*)
{attribute 'reflection'} 
FUNCTION_BLOCK FB_Mitsubishi_MRJ4TM EXTENDS FB_LinkDataReal 
VAR_INPUT
	pControl			: PVOID; //Pocess data from fieldbus, 29 BYTES FROM FIELDBUS
	pStatus				: PVOID; //Pocess data to fieldbus, 41 BYTES FROM FIELDBUS		
	stControl	 		: ST_Mitsubishi_MRJ4TM_Control;
	stConfig			: ST_Mitsubishi_MRJ4TM_Config;
	bSTO 				: BOOL := TRUE;
END_VAR

VAR_OUTPUT
	stStatus 			: ST_Mitsubishi_MRJ4TM_Status;	
END_VAR

VAR		
	{attribute 'instance-path'} 
    {attribute 'noinit'} 
    _sPath 				: STRING;
	_fbStateMachine 	: FB_DS402_FSM;
	_fbEncoder 			: FB_Encoder;	
END_VAR

SUPER^();
InitRun();

GetControlData();
Cycle();
SetStatusData();

METHOD PRIVATE Cycle
IF NOT bSTO THEN RETURN; END_IF

_fbStateMachine.stControl := stControl.nControlWord;
_fbStateMachine();
stStatus.nStatusWord := _fbStateMachine.stStatus;

IF (_fbStateMachine._eState = E_DS402_State.S4_OperationEnabled) THEN	
	
	_fbEncoder.fValue :=  stConfig.fPositionOffset + _fbEncoder.INC_TO_LREAL(stControl.nTargetPosit, 1);
	_fbEncoder();
END_IF

IF stConfig.bSyncOpMode THEN
	stStatus.nStatusWord.b12_OperationModeSpecific := stControl.nControlWord.b4_OperationModeSpecific;
	stStatus.nStatusWord.b13_OperationModeSpecific := stControl.nControlWord.b5_OperationModeSpecific;
	stStatus.nStatusWord.b14_OperationModeSpecific := stControl.nControlWord.b6_OperationModeSpecific;
END_IF


stStatus.nPositionActualValue := _fbEncoder.nResult;
stStatus.nModesOfOperationDisplay := stControl.nModesOfOperation;

//Set Link Data
ControlData := LREAL_TO_REAL(_fbEncoder.fResult);
END_METHOD

PROPERTY eState : E_DS402_State
GET
eState := _fbStateMachine.eState;
END_GET
END_PROPERTY

PROPERTY PUBLIC fbEncoder : REFERENCE TO FB_Encoder
GET
fbEncoder REF= _fbEncoder;
END_GET
END_PROPERTY

METHOD INTERNAL GetControlData
IF pControl <= 0 OR stConfig.bForceMode THEN RETURN; END_IF

(*nModesOfOperation*) 			F_Memcpy(ADR(stControl), pControl, 1, stConfig.bSwapProcessData);
(*nControlWord*)				F_Memcpy(ADR(stControl)+ 1, pControl + 1, 2, stConfig.bSwapProcessData);
(*nControlID1*)					F_Memcpy(ADR(stControl) + 3, pControl + 3, 2, stConfig.bSwapProcessData);
(*nControlID2*)					F_Memcpy(ADR(stControl) + 5, pControl + 5, 2, stConfig.bSwapProcessData);
(*nControlID3*)					F_Memcpy(ADR(stControl) + 7, pControl + 7, 2, stConfig.bSwapProcessData);
(*nTargetPosit*)				F_Memcpy(ADR(stControl) + 9, pControl + 9, 4, stConfig.bSwapProcessData);
(*nTargetVeloc*)				F_Memcpy(ADR(stControl) + 13, pControl + 13, 4, stConfig.bSwapProcessData);
(*nVelocityLimitValue*)			F_Memcpy(ADR(stControl) + 17, pControl + 17, 4, stConfig.bSwapProcessData);
(*nTargetTorque*)				F_Memcpy(ADR(stControl) + 21, pControl + 21, 2, stConfig.bSwapProcessData);
(*nPositiveTorqueLimitValue*)	F_Memcpy(ADR(stControl) + 23, pControl + 23, 2, stConfig.bSwapProcessData);
(*nNegativeTorqueLimitValue*)	F_Memcpy(ADR(stControl) + 25, pControl + 25, 2, stConfig.bSwapProcessData);
(*nTouchProbeFunction*)			F_Memcpy(ADR(stControl) + 27, pControl + 27, 2, stConfig.bSwapProcessData);
END_METHOD

METHOD PRIVATE InitRun
VAR_INST
	bInitRun : BOOL := TRUE;
END_VAR
IF NOT bInitRun THEN RETURN; END_IF
bInitRun := FALSE;

IF pControl = 0 OR pStatus = 0 THEN
	ADSLOGSTR(ADSLOG_MSGTYPE_WARN, '%s', CONCAT(_sPath, ' PLC IO is not assigned!'));	
END_IF
END_METHOD

METHOD INTERNAL SetStatusData
IF pStatus <= 0 THEN RETURN; END_IF

(*nModesOfOperationDisplay*) 	F_Memcpy(pStatus, ADR(stStatus), 1, stConfig.bSwapProcessData);
(*nStatusWord*) 				F_Memcpy(pStatus + 1, ADR(stStatus) + 1, 2, stConfig.bSwapProcessData);
(*nStatusDO1*) 					F_Memcpy(pStatus + 3, ADR(stStatus) + 3, 2, stConfig.bSwapProcessData);
(*nStatusDO2*) 					F_Memcpy(pStatus + 5, ADR(stStatus) + 5, 2, stConfig.bSwapProcessData);
(*nStatusDO3*) 					F_Memcpy(pStatus + 7, ADR(stStatus) + 7, 2, stConfig.bSwapProcessData);
(*nPositionActualValue*) 		F_Memcpy(pStatus + 9, ADR(stStatus) + 9, 4, stConfig.bSwapProcessData);
(*nVelocityActualValue*) 		F_Memcpy(pStatus + 13, ADR(stStatus) + 13, 4, stConfig.bSwapProcessData);
(*nFollowingErrorActualValue*) 	F_Memcpy(pStatus + 17, ADR(stStatus) + 17, 4, stConfig.bSwapProcessData);
(*nTorqueActualValue*) 			F_Memcpy(pStatus + 21, ADR(stStatus) + 21, 2, stConfig.bSwapProcessData);
(*nTouchProbeStatus*) 			F_Memcpy(pStatus + 23, ADR(stStatus) + 23, 2, stConfig.bSwapProcessData);
(*nTouchProbePos1PosValue*) 	F_Memcpy(pStatus + 25, ADR(stStatus) + 25, 4, stConfig.bSwapProcessData);
(*nTouchProbePos1NegValue*) 	F_Memcpy(pStatus + 29, ADR(stStatus) + 29, 4, stConfig.bSwapProcessData);
(*nTouchProbePos2PosValue*) 	F_Memcpy(pStatus + 33, ADR(stStatus) + 33, 4, stConfig.bSwapProcessData);
(*nTouchProbePos2NegValue*) 	F_Memcpy(pStatus + 37, ADR(stStatus) + 37, 4, stConfig.bSwapProcessData);
END_METHOD

END_FUNCTION_BLOCK

// ---- Devices/Terminals/FB_Beckhoff_EK1914.TcPOU
FUNCTION_BLOCK FB_Beckhoff_EK1914
VAR_INPUT
	bSafetyIn1		: BOOL;
	bSafetyIn2		: BOOL;
	bInput0			: BOOL;
	bInput1			: BOOL;
	bInput2			: BOOL;
	bInput3			: BOOL;
END_VAR
VAR_OUTPUT
	bSafetyOut1		: BOOL;
	bSafetyOut2		: BOOL;
	bOutput0		: BOOL;
	bOutput1		: BOOL;
	bOutput2		: BOOL;
	bOutput3		: BOOL;
	bOSafetyLinkedOutput0 : BOOL;
	bOSafetyLinkedOutput1 : BOOL;
END_VAR
VAR
	RxPDO			AT %I* : FSOE_6;
	TxPDO			AT %Q* : FSOE_6;	
	fbFsoeSlave		: FB_FsoeSlave;
	nMasterData		: BYTE := 0;
	nSlaveData		: BYTE := 0;
	
	bOutputDIO0		AT %I* : BOOL;
	bOutputDIO1		AT %I* : BOOL;
	bOutputDIO2		AT %I* : BOOL;
	bOutputDIO3		AT %I* : BOOL;
	bOutputDIOSafetyLinkedOutput0		AT %I* : BOOL;
	bOutputDIOSafetyLinkedOutput1		AT %I* : BOOL;
	bInputDIO0		AT %Q* : BOOL;
	bInputDIO1		AT %Q* : BOOL;
	bInputDIO2		AT %Q* : BOOL;
	bInputDIO3		AT %Q* : BOOL;
END_VAR

nSlaveData.0 := bSafetyIn1;
nSlaveData.1 := bSafetyIn2;
bInputDIO0 := bInput0;
bInputDIO1 := bInput1;
bInputDIO2 := bInput2;
bInputDIO3 := bInput3;

fbFsoeSlave();

bSafetyOut1 := nMasterData.0;
bSafetyOut2 := nMasterData.1;
bOutput0 := bOutputDIO0;
bOutput1 := bOutputDIO1;
bOutput2 := bOutputDIO2;
bOutput3 := bOutputDIO3;
bOSafetyLinkedOutput0 := bOutputDIOSafetyLinkedOutput0;
bOSafetyLinkedOutput1 := bOutputDIOSafetyLinkedOutput1;

METHOD FB_init : BOOL
VAR_INPUT
	bInitRetains 	: BOOL; // if TRUE, the retain variables are initialized (warm start / cold start)
	bInCopyCode 	: BOOL;  // if TRUE, the instance afterwards gets moved into the copy code (online change)
END_VAR
fbFsoeSlave.stConfig.nSlaveAddress := 0;
fbFsoeSlave.stConfig.pFromBus := ADR(RxPDO);
fbFsoeSlave.stConfig.pToBus := ADR(TxPDO);
fbFsoeSlave.stConfig.nSizeMaster := 6;
fbFsoeSlave.stConfig.nSizeSlave := 6;
fbFsoeSlave.stConfig.pMasterData := ADR(nMasterData);
fbFsoeSlave.stConfig.pSlaveData := ADR(nSlaveData);
END_METHOD

END_FUNCTION_BLOCK

// ---- Devices/Terminals/FB_Beckhoff_EJ1918.TcPOU
FUNCTION_BLOCK FB_Beckhoff_EJ1918
VAR_INPUT
	bIn1			: BOOL;
	bIn2			: BOOL;
	bIn3			: BOOL;
	bIn4			: BOOL;
END_VAR
VAR
	RxPDO			AT %I* : FSOE_6;
	TxPDO			AT %Q* : FSOE_7;	
	fbFsoeSlave		: FB_FsoeSlave;
	nMasterData		: BYTE := 0;
	nSlaveData		: WORD := 0;
END_VAR

nSlaveData.0 := bIn1;
nSlaveData.1 := bIn1;
nSlaveData.3 := bIn2;
nSlaveData.4 := bIn2;
nSlaveData.6 := bIn3;
nSlaveData.7 := bIn3;
nSlaveData.9 := bIn4;
nSlaveData.10 := bIn4;

fbFsoeSlave();

METHOD FB_init : BOOL
VAR_INPUT
	bInitRetains 	: BOOL; // if TRUE, the retain variables are initialized (warm start / cold start)
	bInCopyCode 	: BOOL;  // if TRUE, the instance afterwards gets moved into the copy code (online change)
END_VAR
fbFsoeSlave.stConfig.nSlaveAddress := 0;
fbFsoeSlave.stConfig.pFromBus := ADR(RxPDO);
fbFsoeSlave.stConfig.pToBus := ADR(TxPDO);
fbFsoeSlave.stConfig.nSizeMaster := 6;
fbFsoeSlave.stConfig.nSizeSlave := 7;
fbFsoeSlave.stConfig.pMasterData := ADR(nMasterData);
fbFsoeSlave.stConfig.pSlaveData := ADR(nSlaveData);
END_METHOD

END_FUNCTION_BLOCK

// ---- Devices/Terminals/FB_Beckhoff_EL1904.TcPOU
FUNCTION_BLOCK FB_Beckhoff_EL1904
VAR_INPUT
	bIn1			: BOOL;
	bIn2			: BOOL;
	bIn3			: BOOL;
	bIn4			: BOOL;
END_VAR
VAR
	RxPDO			AT %I* : FSOE_6;
	TxPDO			AT %Q* : FSOE_6;	
	fbFsoeSlave		: FB_FsoeSlave;
	nMasterData		: BYTE := 0;
	nSlaveData		: BYTE := 0;
END_VAR

nSlaveData.0 := bIn1;
nSlaveData.1 := bIn2;
nSlaveData.2 := bIn3;
nSlaveData.3 := bIn4;

fbFsoeSlave();

METHOD FB_init : BOOL
VAR_INPUT
	bInitRetains 	: BOOL; // if TRUE, the retain variables are initialized (warm start / cold start)
	bInCopyCode 	: BOOL;  // if TRUE, the instance afterwards gets moved into the copy code (online change)
END_VAR
fbFsoeSlave.stConfig.nSlaveAddress := 0;
fbFsoeSlave.stConfig.pFromBus := ADR(RxPDO);
fbFsoeSlave.stConfig.pToBus := ADR(TxPDO);
fbFsoeSlave.stConfig.nSizeMaster := 6;
fbFsoeSlave.stConfig.nSizeSlave := 6;
fbFsoeSlave.stConfig.pMasterData := ADR(nMasterData);
fbFsoeSlave.stConfig.pSlaveData := ADR(nSlaveData);
END_METHOD

END_FUNCTION_BLOCK

// ---- Devices/Terminals/FB_Beckhoff_EL1918.TcPOU
FUNCTION_BLOCK FB_Beckhoff_EL1918
VAR_INPUT
	bIn1			: BOOL;
	bIn2			: BOOL;
	bIn3			: BOOL;
	bIn4			: BOOL;
	bIn5			: BOOL;
	bIn6			: BOOL;
	bIn7			: BOOL;
	bIn8			: BOOL;
END_VAR
VAR
	RxPDO			AT %I* : FSOE_6;
	TxPDO			AT %Q* : FSOE_7;	
	fbFsoeSlave		: FB_FsoeSlave;
	nMasterData		: BYTE := 0;
	nSlaveData		: WORD := 0;
END_VAR

nSlaveData.0 := bIn1;
nSlaveData.2 := bIn2;
nSlaveData.4 := bIn3;
nSlaveData.6 := bIn4;
nSlaveData.8 := bIn5;
nSlaveData.10 := bIn6;
nSlaveData.12 := bIn7;
nSlaveData.14 := bIn8;

fbFsoeSlave();

METHOD FB_init : BOOL
VAR_INPUT
	bInitRetains 	: BOOL; // if TRUE, the retain variables are initialized (warm start / cold start)
	bInCopyCode 	: BOOL;  // if TRUE, the instance afterwards gets moved into the copy code (online change)
END_VAR
fbFsoeSlave.stConfig.nSlaveAddress := 0;
fbFsoeSlave.stConfig.pFromBus := ADR(RxPDO);
fbFsoeSlave.stConfig.pToBus := ADR(TxPDO);
fbFsoeSlave.stConfig.nSizeMaster := 6;
fbFsoeSlave.stConfig.nSizeSlave := 7;
fbFsoeSlave.stConfig.pMasterData := ADR(nMasterData);
fbFsoeSlave.stConfig.pSlaveData := ADR(nSlaveData);
END_METHOD

END_FUNCTION_BLOCK

// ---- Devices/Terminals/FB_Beckhoff_EL2904.TcPOU
FUNCTION_BLOCK FB_Beckhoff_EL2904
VAR_OUTPUT
	bOut1			: BOOL;
	bOut2			: BOOL;
	bOut3			: BOOL;
	bOut4			: BOOL;	
END_VAR
VAR
	RxPDO			AT %I* : FSOE_6;
	TxPDO			AT %Q* : FSOE_6;	
	fbFsoeSlave		: FB_FsoeSlave;
	nMasterData		: BYTE := 0;
	nSlaveData		: BYTE := 0;
END_VAR

fbFsoeSlave();

bOut1 := nMasterData.0;
bOut2 := nMasterData.1;
bOut3 := nMasterData.2;
bOut4 := nMasterData.3;

METHOD FB_init : BOOL
VAR_INPUT
	bInitRetains 	: BOOL; // if TRUE, the retain variables are initialized (warm start / cold start)
	bInCopyCode 	: BOOL;  // if TRUE, the instance afterwards gets moved into the copy code (online change)
END_VAR
fbFsoeSlave.stConfig.nSlaveAddress := 0;
fbFsoeSlave.stConfig.pFromBus := ADR(RxPDO);
fbFsoeSlave.stConfig.pToBus := ADR(TxPDO);
fbFsoeSlave.stConfig.nSizeMaster := 6;
fbFsoeSlave.stConfig.nSizeSlave := 6;
fbFsoeSlave.stConfig.pMasterData := ADR(nMasterData);
fbFsoeSlave.stConfig.pSlaveData := ADR(nSlaveData);
END_METHOD

END_FUNCTION_BLOCK

// ---- Devices/Terminals/FB_FSOE_19.TcPOU
FUNCTION_BLOCK FB_FSOE_19
VAR_INPUT
	SafetyIn				: ULINT;
END_VAR
VAR_OUTPUT
	SafetyOut				: ULINT;
END_VAR
VAR
	RxPDO			AT %I* 	: FSOE_19;
	TxPDO			AT %Q* 	: FSOE_19;
	fbFsoeSlave				: FB_FsoeSlave;
END_VAR

fbFsoeSlave();

METHOD FB_init : BOOL
VAR_INPUT
	bInitRetains : BOOL; // if TRUE, the retain variables are initialized (warm start / cold start)
	bInCopyCode : BOOL;  // if TRUE, the instance afterwards gets moved into the copy code (online change)
END_VAR
fbFsoeSlave.stConfig.nSlaveAddress := 0;
fbFsoeSlave.stConfig.pFromBus := ADR(RxPDO);
fbFsoeSlave.stConfig.pToBus := ADR(TxPDO);
fbFsoeSlave.stConfig.nSizeMaster := 19;
fbFsoeSlave.stConfig.nSizeSlave := 19;
fbFsoeSlave.stConfig.pMasterData := ADR(SafetyOut);
fbFsoeSlave.stConfig.pSlaveData := ADR(SafetyIn);
END_METHOD

END_FUNCTION_BLOCK
